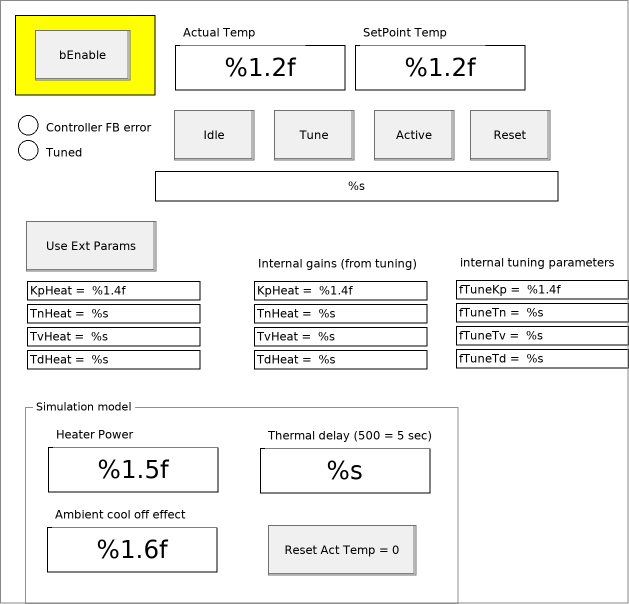
VISUALIZATION HMI  // 629x604
    Rectangle (15,15 140x80), colour toggle: MAIN.bEnabled
    Button (35,30 95x50), "bEnable", pressed state: MAIN.bEnabled
        toggle MAIN.bEnabled
    Rectangle (175,45 170x45), "%1.2f", text variable: MAIN.rTempF, colour toggle: MAIN.bHeaterOn
    Ellipse (18,115 20x20), colour toggle: (MAIN.fbTempContrl.bError) <> 0
    Rectangle (43,115 114x25), "Controller FB error"
    Rectangle (180,20 125x25), "Actual Temp"
    Rectangle (355,45 170x45), "%1.2f", text variable: MAIN.fSetPoint
        OnMouseDown: write the text variable via VisuDialogs.Numpad
    Rectangle (360,20 125x25), "SetPoint Temp"
    Ellipse (18,140 20x20), colour toggle: (MAIN.fbTempContrl.bTuned) <> 0
    Rectangle (43,140 69x25), "Tuned"
    Button (174,110 80x50), "Idle"
        OnMouseUp: execute { MAIN.nControllerMode:=E_CTRL_MODE.eCTRL_MODE_IDLE; }
    Button (274,110 80x50), "Tune"
        OnMouseUp: execute { MAIN.nControllerMode:=E_CTRL_MODE.eCTRL_MODE_TUNE; }
    Button (374,110 80x50), "Active"
        OnMouseUp: execute { MAIN.nControllerMode:=E_CTRL_MODE.eCTRL_MODE_ACTIVE; }
    Rectangle (155,171 403x30), "%s", text variable: MAIN.fbTempContrl.eCtrlState
    Button (26,221 130x50), "Use Ext Params", pressed state: MAIN.stCntrlParam.bSelCtrlParameterSet
        toggle MAIN.stCntrlParam.bSelCtrlParameterSet
    Button (470,110 80x50), "Reset"
        OnMouseUp: execute { MAIN.nControllerMode:=E_CTRL_MODE.eCTRL_MODE_RESET; }
    Rectangle (27,281 173x19), "KpHeat = %1.4f", text variable: MAIN.sParaControlExternal.KpHeat
        OnMouseDown: write the text variable via Edit
    Rectangle (27,304 173x19), "TnHeat = %s", text variable: MAIN.sParaControlExternal.TnHeat
        OnMouseDown: write the text variable via Edit
    Rectangle (27,327 173x19), "TvHeat = %s", text variable: MAIN.sParaControlExternal.TvHeat
        OnMouseDown: write the text variable via Edit
    Rectangle (27,350 173x19), "TdHeat = %s", text variable: MAIN.sParaControlExternal.TdHeat
        OnMouseDown: write the text variable via Edit
    Rectangle (254,281 173x19), "KpHeat = %1.4f", text variable: MAIN.fbTempContrl.sParaControllerInternal.KpHeat
        OnMouseDown: write the text variable via Edit
    Rectangle (254,304 173x19), "TnHeat = %s", text variable: MAIN.fbTempContrl.sParaControllerInternal.TnHeat
        OnMouseDown: write the text variable via Edit
    Rectangle (254,327 173x19), "TvHeat = %s", text variable: MAIN.fbTempContrl.sParaControllerInternal.TvHeat
        OnMouseDown: write the text variable via Edit
    Rectangle (254,350 173x19), "TdHeat = %s", text variable: MAIN.fbTempContrl.sParaControllerInternal.TdHeat
        OnMouseDown: write the text variable via Edit
    Rectangle (255,251 167x25), "Internal gains (from tuning)"
    GroupBox (25,399 433x205), "Simulation model"
        Rectangle (23,48 170x45), "%1.5f", text variable: MAIN.rHeatGain
            OnMouseDown: write the text variable via InputWithLimits, min 0.00001, max 2
        Rectangle (28,23 180x25), "Heater Power"
        Rectangle (235,49 170x45), "%s", text variable: MAIN.iDelay
            OnMouseDown: write the text variable via InputWithLimits, min 1, max 6000
        Rectangle (22,128 170x45), "%1.6f", text variable: MAIN.rCoolOffGain
            OnMouseDown: write the text variable via InputWithLimits, min 0.000001, max 1
        Button (243,126 148x50), "Reset Act Temp = 0", pressed state: MAIN.stCntrlParam.bSelCtrlParameterSet
            toggle MAIN.bResetModel
    Rectangle (265,423 180x25), "Thermal delay (500 = 5 sec)"
    Rectangle (52,502 180x25), "Ambient cool off effect"
    Rectangle (456,280 173x19), "fTuneKp = %1.4f", text variable: MAIN.stCntrlParam.fTuneKp
        OnMouseDown: write the text variable via Edit
    Rectangle (456,303 173x19), "fTuneTn = %s", text variable: MAIN.stCntrlParam.fTuneTn
        OnMouseDown: write the text variable via Edit
    Rectangle (456,326 173x19), "fTuneTv = %s", text variable: MAIN.stCntrlParam.fTuneTv
        OnMouseDown: write the text variable via Edit
    Rectangle (456,349 173x19), "fTuneTd = %s", text variable: MAIN.stCntrlParam.fTuneTd
        OnMouseDown: write the text variable via Edit
    Rectangle (457,250 167x25), "internal tuning parameters"
END_VISUALIZATION

(* stored: Version 1.1.0.1, ProductVersion 3.1.4024.11
   Visu HMI: Id {8ad2170f-4c2b-4822-a55d-798f31eeaa7a} *)
